// TIA Portal V20 export
DATA_BLOCK "InstCallEquipment"   // DB137
{ DB_Accessible_From_OPC_UA := 'FALSE' }
AUTHOR : ERsystem_FA2_DH. Kim
// stored: AssignedProDiagFB Unit1.Em7.ProDiag, DBAccessibleFromOPCUA false, DBAccessibleFromWebserver false, InstanceOfName Unit1.Em7.CallEquipment, InstanceOfType FB, Namespace Unit1.Em7
"Unit1.Em7.CallEquipment"
   // VAR_INPUT
   //    ZoneOperationEnable { ExternalWritable := 'False'} : "LWONIK_typeSafetyZoneManualOperation";
   // END_VAR
   // VAR_IN_OUT
   //    unitStatus : "LAF_typeUnitStatus";
   //    emFeedback : "LUC_typeEmFeedback";
   //    unitAlarmDB : "LAF_typeAlarms";
   // END_VAR
   // VAR
   //    instSequenceSepaClamp { ExternalAccessible := 'False'; ExternalVisible := 'False'; ExternalWritable := 'False'} : "Unit1.Em7.Sequence_1_SepaClamp";
   //    instSequenceSepaGripper { ExternalAccessible := 'False'; ExternalVisible := 'False'; ExternalWritable := 'False'} : "Unit1.Em7.Sequence_2_SepaGripper";
   //    instSequenceJellyRollWinder { ExternalAccessible := 'False'; ExternalVisible := 'False'; ExternalWritable := 'False'} : "Unit1.Em7.Sequence_3_JellyRollWinder";
   //    instSepaClampHomeJob1 { S7_SetPoint := 'True'} : "LAF_SelectJob";
   //    instSepaClampLoadJob2 { S7_SetPoint := 'True'} : "LAF_SelectJob";
   //    instSepaClampUnloadJob3 { S7_SetPoint := 'True'} : "LAF_SelectJob";
   //    instSepaClampUnloadCamJob10 { S7_SetPoint := 'True'} : "LAF_SelectJob";
   //    instSepaClampUnloadStopSyncJob11 { S7_SetPoint := 'True'} : "LAF_SelectJob";
   //    instSepaClampUnloadReturnJob12 { S7_SetPoint := 'True'} : "LAF_SelectJob";
   //    instSepaGripperHomeJob1 { S7_SetPoint := 'True'} : "LAF_SelectJob";
   //    instSepaGripperGripReadyJob2 { S7_SetPoint := 'True'} : "LAF_SelectJob";
   //    instSepaGripperGripSepaTailJob3 { S7_SetPoint := 'True'} : "LAF_SelectJob";
   //    instSepaGripperWinderMoveJob4 { S7_SetPoint := 'True'} : "LAF_SelectJob";
   //    instSepaGripperJellyRollUnGripJob5 { S7_SetPoint := 'True'} : "LAF_SelectJob";
   //    instSepaGripperJellyRollGripJob6 { S7_SetPoint := 'True'} : "LAF_SelectJob";
   //    instSepaGripperUnloadReadyJob7 { S7_SetPoint := 'True'} : "LAF_SelectJob";
   //    instSepaGripperUnloadJob8 { S7_SetPoint := 'True'} : "LAF_SelectJob";
   //    instSepaGripperReturnJob9 { S7_SetPoint := 'True'} : "LAF_SelectJob";
   //    instSepaGripperGripReadyJob11 { S7_SetPoint := 'True'} : "LAF_SelectJob";
   //    instSepaGripperLoadToStackTableJob12 { S7_SetPoint := 'True'} : "LAF_SelectJob";
   //    instSepaGripperUnLoadToJellyRollWinderJob14 { S7_SetPoint := 'True'} : "LAF_SelectJob";
   //    instSepaGripperLoadToJellyRollWinderJob15 { S7_SetPoint := 'True'} : "LAF_SelectJob";
   //    instSepaGripperUnloadToInspectionJob17 { S7_SetPoint := 'True'} : "LAF_SelectJob";
   //    instSepaGripperReturnJob18 { S7_SetPoint := 'True'} : "LAF_SelectJob";
   //    instJellyRollWinderHomeJob1 { S7_SetPoint := 'True'} : "LAF_SelectJob";
   //    instJellyRollWinderLoadJob2 { S7_SetPoint := 'True'} : "LAF_SelectJob";
   //    instJellyRollWinderWinding1Job3 { S7_SetPoint := 'True'} : "LAF_SelectJob";
   //    instJellyRollWinderPusherReadyJob4 { S7_SetPoint := 'True'} : "LAF_SelectJob";
   //    instJellyRollWinderWinding2Job5 { S7_SetPoint := 'True'} : "LAF_SelectJob";
   //    instJellyRollWinderUnloadJob6 { S7_SetPoint := 'True'} : "LAF_SelectJob";
   //    instJellyRollWinderCamWinding1stJob10 { S7_SetPoint := 'True'} : "LAF_SelectJob";
   //    instJellyRollWinderCamPusherReadyJob11 { S7_SetPoint := 'True'} : "LAF_SelectJob";
   //    instJellyRollWinderCamStartSyncJob12 { S7_SetPoint := 'True'} : "LAF_SelectJob";
   //    instJellyRollWinderCamWinding2ndJob13 { S7_SetPoint := 'True'} : "LAF_SelectJob";
   //    instJellyRollWinderCamStopSyncJob14 { S7_SetPoint := 'True'} : "LAF_SelectJob";
   //    instCmSepaClampDetectSensor { ExternalAccessible := 'False'; ExternalVisible := 'False'; ExternalWritable := 'False'} : "LBC_DigitalSignalCn";
   //    instCmSepaGripperDetectSensor { ExternalAccessible := 'False'; ExternalVisible := 'False'; ExternalWritable := 'False'} : "LBC_DigitalSignalCn";
   //    instCmJrWinderDetectSensor { ExternalAccessible := 'False'; ExternalVisible := 'False'; ExternalWritable := 'False'} : "LBC_DigitalSignalCn";
   //    instCmSepaElectrodeDetectSensor { ExternalAccessible := 'False'; ExternalVisible := 'False'; ExternalWritable := 'False'} : "LBC_DigitalSignalCn";
   //    instCmSepaClampSafetyPinDetectSensor { ExternalAccessible := 'False'; ExternalVisible := 'False'; ExternalWritable := 'False'} : "LBC_DigitalSignalCn";
   //    instCmSepaGripperSafetyPinDetectSensor { ExternalAccessible := 'False'; ExternalVisible := 'False'; ExternalWritable := 'False'} : "LBC_DigitalSignalCn";
   //    instCmSepaClampnCutterAxisX { ExternalAccessible := 'False'; ExternalVisible := 'False'; ExternalWritable := 'False'} : "LBC_Axis64Pos_TecPlcCn";
   //    instCmSepaClampnCutterAxisZ { ExternalAccessible := 'False'; ExternalVisible := 'False'; ExternalWritable := 'False'} : "LBC_Axis64Pos_TecPlcCn";
   //    instCmSepaGripperAxisX { ExternalAccessible := 'False'; ExternalVisible := 'False'; ExternalWritable := 'False'} : "LBC_Axis64Pos_TecPlcCn";
   //    instCmSepaGripperAxisZ { ExternalAccessible := 'False'; ExternalVisible := 'False'; ExternalWritable := 'False'} : "LBC_Axis64Pos_TecPlcCn";
   //    instCmSepaGripperAxisC { ExternalAccessible := 'False'; ExternalVisible := 'False'; ExternalWritable := 'False'} : "LBC_Axis64Pos_TecPlcCn";
   //    instCmJRWinderRearAxisY { ExternalAccessible := 'False'; ExternalVisible := 'False'; ExternalWritable := 'False'} : "LBC_Axis64Pos_TecPlcCn";
   //    instCmJRWinderFrontAxisY { ExternalAccessible := 'False'; ExternalVisible := 'False'; ExternalWritable := 'False'} : "LBC_Axis64Pos_TecPlcCn";
   //    instCmJRWinderAxisB { ExternalAccessible := 'False'; ExternalVisible := 'False'; ExternalWritable := 'False'} : "LBC_Axis64Pos_TecPlcCn";
   //    instCmJRPusherAxisZ { ExternalAccessible := 'False'; ExternalVisible := 'False'; ExternalWritable := 'False'} : "LBC_Axis64Pos_TecPlcCn";
   //    instInterlockSepaClampnCutterAxisX { S7_SetPoint := 'True'} : "LER_Axis64Pos_InterlockSummary";
   //    instInterlockSepaClampnCutterAxisZ { S7_SetPoint := 'True'} : "LER_Axis64Pos_InterlockSummary";
   //    instInterlockSepaGripperAxisX { S7_SetPoint := 'True'} : "LER_Axis64Pos_InterlockSummary";
   //    instInterlockSepaGripperAxisZ { S7_SetPoint := 'True'} : "LER_Axis64Pos_InterlockSummary";
   //    instInterlockSepaGripperAxisC { S7_SetPoint := 'True'} : "LER_Axis64Pos_InterlockSummary";
   //    instInterlockJRWinderRearAxisY { S7_SetPoint := 'True'} : "LER_Axis64Pos_InterlockSummary";
   //    instInterlockJRWinderFrontAxisY { S7_SetPoint := 'True'} : "LER_Axis64Pos_InterlockSummary";
   //    instInterlockJRWinderAxisB { S7_SetPoint := 'True'} : "LER_Axis64Pos_InterlockSummary";
   //    instInterlockJRPusherAxisZ { S7_SetPoint := 'True'} : "LER_Axis64Pos_InterlockSummary";
   //    instSepaClampAxisXCalculateCam { S7_SetPoint := 'True'} : "Unit1.Em7.SepaClampXCalculateCam";
   //    instSepaClampAxisZCalculateCam { S7_SetPoint := 'True'} : "Unit1.Em7.SepaClampZCalculateCam";
   //    instJRPusherAxisZCalculateCam { S7_SetPoint := 'True'} : "Unit1.Em7.PusherRollerZCalculateCam";
   //    instSepaClampAxisXMCCamIn { S7_SetPoint := 'True'} : MC_CAMIN;
   //    instSepaClampAxisZMCCamIn { S7_SetPoint := 'True'} : MC_CAMIN;
   //    instJRPusherAxisZMCCamIn { S7_SetPoint := 'True'} : MC_CAMIN;
   //    instCmSepaCutterUpDown { ExternalAccessible := 'False'; ExternalVisible := 'False'; ExternalWritable := 'False'} : "LBC_TwoWayActuatorCn";
   //    instCmSepaClampTopUpDown { ExternalAccessible := 'False'; ExternalVisible := 'False'; ExternalWritable := 'False'} : "LBC_TwoWayActuatorCn";
   //    instCmSepaClampBottomUpDown { ExternalAccessible := 'False'; ExternalVisible := 'False'; ExternalWritable := 'False'} : "LBC_TwoWayActuatorCn";
   //    instCmStackGripperOpenClose { ExternalAccessible := 'False'; ExternalVisible := 'False'; ExternalWritable := 'False'} : "LBC_TwoWayActuatorCn";
   //    instCmStackGripperFwdBwd { ExternalAccessible := 'False'; ExternalVisible := 'False'; ExternalWritable := 'False'} : "LBC_TwoWayActuatorCn";
   //    instCmJRWinderClampTopRearUpDown { ExternalAccessible := 'False'; ExternalVisible := 'False'; ExternalWritable := 'False'} : "LBC_TwoWayActuatorCn";
   //    instCmJRWinderClampBtmRearUpDown { ExternalAccessible := 'False'; ExternalVisible := 'False'; ExternalWritable := 'False'} : "LBC_TwoWayActuatorCn";
   //    instCmJRWinderClampTopFrontUpDown { ExternalAccessible := 'False'; ExternalVisible := 'False'; ExternalWritable := 'False'} : "LBC_TwoWayActuatorCn";
   //    instCmJRWinderClampBtmFrontUpDown { ExternalAccessible := 'False'; ExternalVisible := 'False'; ExternalWritable := 'False'} : "LBC_TwoWayActuatorCn";
   //    instCmPusherRollerFwdBwd { ExternalAccessible := 'False'; ExternalVisible := 'False'; ExternalWritable := 'False'} : "LBC_TwoWayActuatorCn";
   //    instManageAlarms { ExternalAccessible := 'False'; ExternalVisible := 'False'; ExternalWritable := 'False'} : "LAF_ManageAlarms";
   //    instEventsPFE { ExternalAccessible := 'False'; ExternalVisible := 'False'; ExternalWritable := 'False'} : "Unit1.Em7.EventsPFE";
   //    instLER_BrakeTestSepaClampNCutterAxisZ : "LER_BrakeTest";
   //    instLER_BrakeTestSepaGripperAxisZ { S7_SetPoint := 'True'} : "LER_BrakeTest";
   //    instLER_BrakeTestJRPusherAxisZ { S7_SetPoint := 'True'} : "LER_BrakeTest";
   //    statUnitStatus { ExternalAccessible := 'False'; ExternalVisible := 'False'; ExternalWritable := 'False'} : "LAF_typeUnitStatus";
   //    statSlmStatus : Struct
   //       running { ExternalWritable := 'False'} : Bool;
   //       powerOff { ExternalWritable := 'False'} : Bool;
   //    END_STRUCT;
   //    statAllBrakeTest { ExternalWritable := 'False'} : "LER_typeBrakeTestUnitCommands";
   //    statTonTime { ExternalAccessible := 'False'; ExternalVisible := 'False'; ExternalWritable := 'False'} : Array[0..1999] of TON_TIME;
   //    statTofTime { ExternalAccessible := 'False'; ExternalVisible := 'False'; ExternalWritable := 'False'} : Array[0..99] of TOF_TIME;
   //    statPulse { ExternalAccessible := 'False'; ExternalVisible := 'False'; ExternalWritable := 'False'} : Struct
   //       miscellaneous : Array[0..99] of Bool;
   //       workingDone : Struct
   //          sepaClamp : Array[0..99] of Bool;
   //          sepaGripper : Array[0..99] of Bool;
   //          winder : Array[0..99] of Bool;
   //       END_STRUCT;
   //       axisEnable : Array[0..99] of Bool;
   //       brakeTest : Array[0..99] of Bool;
   //    END_STRUCT;
   //    statEnableManualCmds { ExternalAccessible := 'False'; ExternalVisible := 'False'; ExternalWritable := 'False'} : Bool;
   //    scan_on : Bool;
   //    "*** Interlock Axis ***" { ExternalAccessible := 'False'; ExternalVisible := 'False'; ExternalWritable := 'False'} : Bool;
   //    instSepaClampnCutterAxisX_CW { S7_SetPoint := 'True'} : "Jog.LER_Axis";
   //    instSepaClampnCutterAxisX_CCW { S7_SetPoint := 'True'} : "Jog.LER_Axis";
   //    instSepaClampnCutterAxisX_Home { S7_SetPoint := 'True'} : "Homing.LER_Axis";
   //    instSepaClampnCutterAxisX_Position { S7_SetPoint := 'True'} : Array[0..6] of "Position.LER_Axis";
   //    instSepaClampnCutterAxisZ_CW { S7_SetPoint := 'True'} : "Jog.LER_Axis";
   //    instSepaClampnCutterAxisZ_CCW { S7_SetPoint := 'True'} : "Jog.LER_Axis";
   //    instSepaClampnCutterAxisZ_Home { S7_SetPoint := 'True'} : "Homing.LER_Axis";
   //    instSepaClampnCutterAxisZ_Position { S7_SetPoint := 'True'} : Array[0..6] of "Position.LER_Axis";
   //    instSepaGripperAxisX_CW { S7_SetPoint := 'True'} : "Jog.LER_Axis";
   //    instSepaGripperAxisX_CCW { S7_SetPoint := 'True'} : "Jog.LER_Axis";
   //    instSepaGripperAxisX_Home { S7_SetPoint := 'True'} : "Homing.LER_Axis";
   //    instSepaGripperAxisX_Position { S7_SetPoint := 'True'} : Array[0..15] of "Position.LER_Axis";
   //    instSepaGripperAxisZ_CW { S7_SetPoint := 'True'} : "Jog.LER_Axis";
   //    instSepaGripperAxisZ_CCW { S7_SetPoint := 'True'} : "Jog.LER_Axis";
   //    instSepaGripperAxisZ_Home { S7_SetPoint := 'True'} : "Homing.LER_Axis";
   //    instSepaGripperAxisZ_Position { S7_SetPoint := 'True'} : Array[0..6] of "Position.LER_Axis";
   //    instSepaGripperAxisC_CW { S7_SetPoint := 'True'} : "Jog.LER_Axis";
   //    instSepaGripperAxisC_CCW { S7_SetPoint := 'True'} : "Jog.LER_Axis";
   //    instSepaGripperAxisC_Home { S7_SetPoint := 'True'} : "Homing.LER_Axis";
   //    instSepaGripperAxisC_Position { S7_SetPoint := 'True'} : Array[0..6] of "Position.LER_Axis";
   //    instJRWinderRearAxisY_CW { S7_SetPoint := 'True'} : "Jog.LER_Axis";
   //    instJRWinderRearAxisY_CCW { S7_SetPoint := 'True'} : "Jog.LER_Axis";
   //    instJRWinderRearAxisY_Home { S7_SetPoint := 'True'} : "Homing.LER_Axis";
   //    instJRWinderRearAxisY_Position { S7_SetPoint := 'True'} : Array[0..6] of "Position.LER_Axis";
   //    instJRWinderFrontAxisY_CW { S7_SetPoint := 'True'} : "Jog.LER_Axis";
   //    instJRWinderFrontAxisY_CCW { S7_SetPoint := 'True'} : "Jog.LER_Axis";
   //    instJRWinderFrontAxisY_Home { S7_SetPoint := 'True'} : "Homing.LER_Axis";
   //    instJRWinderFrontAxisY_Position { S7_SetPoint := 'True'} : Array[0..6] of "Position.LER_Axis";
   //    instJRWinderAxisB_CW { S7_SetPoint := 'True'} : "Jog.LER_Axis";
   //    instJRWinderAxisB_CCW { S7_SetPoint := 'True'} : "Jog.LER_Axis";
   //    instJRWinderAxisB_Home { S7_SetPoint := 'True'} : "Homing.LER_Axis";
   //    instJRWinderAxisB_Position { S7_SetPoint := 'True'} : Array[0..8] of "Position.LER_Axis";
   //    instJRPusherAxisZ_CW { S7_SetPoint := 'True'} : "Jog.LER_Axis";
   //    instJRPusherAxisZ_CCW { S7_SetPoint := 'True'} : "Jog.LER_Axis";
   //    instJRPusherAxisZ_Home { S7_SetPoint := 'True'} : "Homing.LER_Axis";
   //    instJRPusherAxisZ_Position { S7_SetPoint := 'True'} : Array[0..6] of "Position.LER_Axis";
   //    "*** Interlock Actuator ******" { ExternalAccessible := 'False'; ExternalVisible := 'False'; ExternalWritable := 'False'} : Bool;
   //    instCmSepaCutterUpDownInterlock : Array[0..1] of "Cylinder.LER_Actuator";
   //    instCmSepaClampTopUpDownInterlock { S7_SetPoint := 'True'} : Array[0..1] of "Cylinder.LER_Actuator";
   //    instCmSepaClampBottomUpDownInterlock { S7_SetPoint := 'True'} : Array[0..1] of "Cylinder.LER_Actuator";
   //    instCmStackGripperOpenCloseInterlock { S7_SetPoint := 'True'} : Array[0..1] of "Cylinder.LER_Actuator";
   //    instCmStackGripperFwdBwdInterlock { S7_SetPoint := 'True'} : Array[0..1] of "Cylinder.LER_Actuator";
   //    instCmJRWinderClampTopRearUpDownInterlock { S7_SetPoint := 'True'} : Array[0..1] of "Cylinder.LER_Actuator";
   //    instCmJRWinderClampBtmRearUpDownInterlock { S7_SetPoint := 'True'} : Array[0..1] of "Cylinder.LER_Actuator";
   //    instCmJRWinderClampTopFrontUpDownInterlock { S7_SetPoint := 'True'} : Array[0..1] of "Cylinder.LER_Actuator";
   //    instCmJRWinderClampBtmFrontUpDownInterlock { S7_SetPoint := 'True'} : Array[0..1] of "Cylinder.LER_Actuator";
   //    instCmPusherRollerFwdBwdInterlock { S7_SetPoint := 'True'} : Array[0..1] of "Cylinder.LER_Actuator";
   //    Tracking_07 { S7_SetPoint := 'True'} : "Unit1.Em7.PartData";
   //    AXIS34 : "LER_CM_Name";
   //    AXIS39 : "LER_CM_Name";
   //    Cylinder38 : "LER_CM_Name";
   //    Cylinder43 : "LER_CM_Name";
   //    citi_Ptrig : Array[0..20] of Bool;
   //    citiTon : Array[0..20] of TON_TIME;
   //    citi : Time;
   //    citiTest : Array[0..20] of Bool;
   // END_VAR
BEGIN
   ZoneOperationEnable.autoStartEnable := FALSE;
   ZoneOperationEnable.doorLockEnable := TRUE;
   ZoneOperationEnable.doorUnlockEnable := TRUE;
   ZoneOperationEnable.rc_AutoEnable := FALSE;
   ZoneOperationEnable.rc_RollChangeEnable := FALSE;
   ZoneOperationEnable.rc_DoorLockEnable := TRUE;
   ZoneOperationEnable.rc_DoorUnlockEnable := TRUE;
   ZoneOperationEnable.hmiOperationEnable := TRUE;
   ZoneOperationEnable.phmiOperationEnable := FALSE;
   instSequenceSepaClamp.statSelectedJobNumber := 0;
   instSequenceSepaClamp.instSequenceLADStatus.parentReferenceDesignator := WSTRING#'';
   instSequenceSepaClamp.instSequenceLADStatus.idleStep := 1;
   instSequenceSepaClamp.instSequenceLADStatus.stoppedStep := 9001;
   instSequenceSepaClamp.instSequenceLADStatus.setJobNumber := 0;
   instSequenceSepaClamp.instSequenceLADStatus.activeJobNumber := 0;
   instSequenceSepaClamp.instSequenceLADStatus.previousCycleJobNumber := 0;
   instSequenceSepaClamp.instSequenceLADStatus.statCurrentJob := 0;
   instSequenceSepaClamp.instSequenceLADStatus.statStepComplete := FALSE;
   instSequenceSepaClamp.instSequenceLADControl.idleStep := 1;
   instSequenceSepaClamp.instSequenceLADControl.stoppedStep := 9001;
   instSequenceSepaClamp.instSequenceLADControl.resetJobs := FALSE;
   instSequenceSepaClamp.instSequenceLADControl.statMemInit := FALSE;
   instSequenceSepaClamp.instSequenceLADControl.statMemImmediateStop := FALSE;
   instSequenceSepaClamp.instSequenceLADControl.statMemNextStep1 := FALSE;
   instSequenceSepaClamp.instSequenceLADControl.statMemNextStep2 := FALSE;
   instSequenceSepaClamp.instSequenceLADControl.statMemNextStep3 := FALSE;
   instSequenceSepaClamp.instSequenceLADControl.statFirstCycleInit := FALSE;
   instCmSepaClampDetectSensor.enable := TRUE;
   instCmSepaClampDetectSensor.parentReferenceDesignator := WSTRING#'';
   instCmSepaClampDetectSensor.digitalValue := FALSE;
   instCmSepaClampDetectSensor.simulatedDigitalValue := FALSE;
   instCmSepaClampDetectSensor.statProcessValues.enable := TRUE;
   instCmSepaClampDetectSensor.statProcessValues.referenceDesignator := WSTRING#'DigitalSignal';
   instCmSepaClampDetectSensor.statProcessValues.simulation := FALSE;
   instCmSepaClampDetectSensor.statProcessValues.processValue := FALSE;
   instCmSepaClampDetectSensor.statProcessValues.error := FALSE;
   instCmSepaClampDetectSensor.statProcessValues.status := 16#0000;
   instCmSepaClampDetectSensor.statDiagnostics.status := 16#0000;
   instCmSepaClampDetectSensor.statDiagnostics.subfunctionStatus := 16#0000;
   instCmSepaClampDetectSensor.statDiagnostics.stateNumber := 0;
   instCmSepaClampDetectSensor.statEmptyDiagnostics.status := 16#0000;
   instCmSepaClampDetectSensor.statEmptyDiagnostics.subfunctionStatus := 16#0000;
   instCmSepaClampDetectSensor.statEmptyDiagnostics.stateNumber := 0;
   instCmSepaClampDetectSensor.instOnDelay.PT := T#0MS;
   instCmSepaClampDetectSensor.instOnDelay.IN := FALSE;
   instCmSepaClampDetectSensor.instOffDelay.PT := T#0MS;
   instCmSepaClampDetectSensor.instOffDelay.IN := FALSE;
   instCmSepaClampDetectSensor.statDisableAlarms := FALSE;
   instCmSepaClampDetectSensor.statErrorState := 16#0000;
   instCmSepaClampDetectSensor.statFirstCall := FALSE;
   instCmSepaClampDetectSensor.statResetPrevious := FALSE;
   instCmSepaClampDetectSensor.statEnablePrevious := TRUE;
   instCmSepaClampDetectSensor.statProcessValuePrevious := FALSE;
   instCmSepaGripperDetectSensor.enable := TRUE;
   instCmSepaGripperDetectSensor.parentReferenceDesignator := WSTRING#'';
   instCmSepaGripperDetectSensor.digitalValue := TRUE;
   instCmSepaGripperDetectSensor.simulatedDigitalValue := FALSE;
   instCmSepaGripperDetectSensor.statProcessValues.enable := TRUE;
   instCmSepaGripperDetectSensor.statProcessValues.referenceDesignator := WSTRING#'DigitalSignal';
   instCmSepaGripperDetectSensor.statProcessValues.simulation := FALSE;
   instCmSepaGripperDetectSensor.statProcessValues.processValue := TRUE;
   instCmSepaGripperDetectSensor.statProcessValues.error := FALSE;
   instCmSepaGripperDetectSensor.statProcessValues.status := 16#0000;
   instCmSepaGripperDetectSensor.statDiagnostics.status := 16#0000;
   instCmSepaGripperDetectSensor.statDiagnostics.subfunctionStatus := 16#0000;
   instCmSepaGripperDetectSensor.statDiagnostics.stateNumber := 0;
   instCmSepaGripperDetectSensor.statEmptyDiagnostics.status := 16#0000;
   instCmSepaGripperDetectSensor.statEmptyDiagnostics.subfunctionStatus := 16#0000;
   instCmSepaGripperDetectSensor.statEmptyDiagnostics.stateNumber := 0;
   instCmSepaGripperDetectSensor.instOnDelay.PT := T#0MS;
   instCmSepaGripperDetectSensor.instOnDelay.IN := FALSE;
   instCmSepaGripperDetectSensor.instOffDelay.PT := T#0MS;
   instCmSepaGripperDetectSensor.instOffDelay.IN := FALSE;
   instCmSepaGripperDetectSensor.statDisableAlarms := FALSE;
   instCmSepaGripperDetectSensor.statErrorState := 16#0000;
   instCmSepaGripperDetectSensor.statFirstCall := FALSE;
   instCmSepaGripperDetectSensor.statResetPrevious := FALSE;
   instCmSepaGripperDetectSensor.statEnablePrevious := TRUE;
   instCmSepaGripperDetectSensor.statProcessValuePrevious := TRUE;
   instCmJrWinderDetectSensor.enable := TRUE;
   instCmJrWinderDetectSensor.parentReferenceDesignator := WSTRING#'';
   instCmJrWinderDetectSensor.digitalValue := FALSE;
   instCmJrWinderDetectSensor.simulatedDigitalValue := FALSE;
   instCmJrWinderDetectSensor.statProcessValues.enable := TRUE;
   instCmJrWinderDetectSensor.statProcessValues.referenceDesignator := WSTRING#'DigitalSignal';
   instCmJrWinderDetectSensor.statProcessValues.simulation := FALSE;
   instCmJrWinderDetectSensor.statProcessValues.processValue := FALSE;
   instCmJrWinderDetectSensor.statProcessValues.error := FALSE;
   instCmJrWinderDetectSensor.statProcessValues.status := 16#0000;
   instCmJrWinderDetectSensor.statDiagnostics.status := 16#0000;
   instCmJrWinderDetectSensor.statDiagnostics.subfunctionStatus := 16#0000;
   instCmJrWinderDetectSensor.statDiagnostics.stateNumber := 0;
   instCmJrWinderDetectSensor.statEmptyDiagnostics.status := 16#0000;
   instCmJrWinderDetectSensor.statEmptyDiagnostics.subfunctionStatus := 16#0000;
   instCmJrWinderDetectSensor.statEmptyDiagnostics.stateNumber := 0;
   instCmJrWinderDetectSensor.instOnDelay.PT := T#0MS;
   instCmJrWinderDetectSensor.instOnDelay.IN := FALSE;
   instCmJrWinderDetectSensor.instOffDelay.PT := T#0MS;
   instCmJrWinderDetectSensor.instOffDelay.IN := FALSE;
   instCmJrWinderDetectSensor.statDisableAlarms := FALSE;
   instCmJrWinderDetectSensor.statErrorState := 16#0000;
   instCmJrWinderDetectSensor.statFirstCall := FALSE;
   instCmJrWinderDetectSensor.statResetPrevious := FALSE;
   instCmJrWinderDetectSensor.statEnablePrevious := TRUE;
   instCmJrWinderDetectSensor.statProcessValuePrevious := FALSE;
   instCmSepaElectrodeDetectSensor.enable := TRUE;
   instCmSepaElectrodeDetectSensor.parentReferenceDesignator := WSTRING#'';
   instCmSepaElectrodeDetectSensor.digitalValue := FALSE;
   instCmSepaElectrodeDetectSensor.simulatedDigitalValue := FALSE;
   instCmSepaElectrodeDetectSensor.statProcessValues.enable := TRUE;
   instCmSepaElectrodeDetectSensor.statProcessValues.referenceDesignator := WSTRING#'DigitalSignal';
   instCmSepaElectrodeDetectSensor.statProcessValues.simulation := FALSE;
   instCmSepaElectrodeDetectSensor.statProcessValues.processValue := FALSE;
   instCmSepaElectrodeDetectSensor.statProcessValues.error := FALSE;
   instCmSepaElectrodeDetectSensor.statProcessValues.status := 16#0000;
   instCmSepaElectrodeDetectSensor.statDiagnostics.status := 16#0000;
   instCmSepaElectrodeDetectSensor.statDiagnostics.subfunctionStatus := 16#0000;
   instCmSepaElectrodeDetectSensor.statDiagnostics.stateNumber := 0;
   instCmSepaElectrodeDetectSensor.statEmptyDiagnostics.status := 16#0000;
   instCmSepaElectrodeDetectSensor.statEmptyDiagnostics.subfunctionStatus := 16#0000;
   instCmSepaElectrodeDetectSensor.statEmptyDiagnostics.stateNumber := 0;
   instCmSepaElectrodeDetectSensor.instOnDelay.PT := T#0MS;
   instCmSepaElectrodeDetectSensor.instOnDelay.IN := FALSE;
   instCmSepaElectrodeDetectSensor.instOffDelay.PT := T#0MS;
   instCmSepaElectrodeDetectSensor.instOffDelay.IN := FALSE;
   instCmSepaElectrodeDetectSensor.statDisableAlarms := FALSE;
   instCmSepaElectrodeDetectSensor.statErrorState := 16#0000;
   instCmSepaElectrodeDetectSensor.statFirstCall := FALSE;
   instCmSepaElectrodeDetectSensor.statResetPrevious := FALSE;
   instCmSepaElectrodeDetectSensor.statEnablePrevious := TRUE;
   instCmSepaElectrodeDetectSensor.statProcessValuePrevious := FALSE;
   instCmSepaClampSafetyPinDetectSensor.enable := TRUE;
   instCmSepaClampSafetyPinDetectSensor.parentReferenceDesignator := WSTRING#'';
   instCmSepaClampSafetyPinDetectSensor.digitalValue := TRUE;
   instCmSepaClampSafetyPinDetectSensor.simulatedDigitalValue := FALSE;
   instCmSepaClampSafetyPinDetectSensor.statProcessValues.enable := TRUE;
   instCmSepaClampSafetyPinDetectSensor.statProcessValues.referenceDesignator := WSTRING#'DigitalSignal';
   instCmSepaClampSafetyPinDetectSensor.statProcessValues.simulation := FALSE;
   instCmSepaClampSafetyPinDetectSensor.statProcessValues.processValue := TRUE;
   instCmSepaClampSafetyPinDetectSensor.statProcessValues.error := FALSE;
   instCmSepaClampSafetyPinDetectSensor.statProcessValues.status := 16#0000;
   instCmSepaClampSafetyPinDetectSensor.statDiagnostics.status := 16#0000;
   instCmSepaClampSafetyPinDetectSensor.statDiagnostics.subfunctionStatus := 16#0000;
   instCmSepaClampSafetyPinDetectSensor.statDiagnostics.stateNumber := 0;
   instCmSepaClampSafetyPinDetectSensor.statEmptyDiagnostics.status := 16#0000;
   instCmSepaClampSafetyPinDetectSensor.statEmptyDiagnostics.subfunctionStatus := 16#0000;
   instCmSepaClampSafetyPinDetectSensor.statEmptyDiagnostics.stateNumber := 0;
   instCmSepaClampSafetyPinDetectSensor.instOnDelay.PT := T#0MS;
   instCmSepaClampSafetyPinDetectSensor.instOnDelay.IN := FALSE;
   instCmSepaClampSafetyPinDetectSensor.instOffDelay.PT := T#0MS;
   instCmSepaClampSafetyPinDetectSensor.instOffDelay.IN := FALSE;
   instCmSepaClampSafetyPinDetectSensor.statDisableAlarms := FALSE;
   instCmSepaClampSafetyPinDetectSensor.statErrorState := 16#0000;
   instCmSepaClampSafetyPinDetectSensor.statFirstCall := FALSE;
   instCmSepaClampSafetyPinDetectSensor.statResetPrevious := FALSE;
   instCmSepaClampSafetyPinDetectSensor.statEnablePrevious := TRUE;
   instCmSepaClampSafetyPinDetectSensor.statProcessValuePrevious := TRUE;
   instCmSepaGripperSafetyPinDetectSensor.enable := FALSE;
   instCmSepaGripperSafetyPinDetectSensor.parentReferenceDesignator := WSTRING#'';
   instCmSepaGripperSafetyPinDetectSensor.digitalValue := FALSE;
   instCmSepaGripperSafetyPinDetectSensor.simulatedDigitalValue := FALSE;
   instCmSepaGripperSafetyPinDetectSensor.statProcessValues.enable := FALSE;
   instCmSepaGripperSafetyPinDetectSensor.statProcessValues.referenceDesignator := WSTRING#'';
   instCmSepaGripperSafetyPinDetectSensor.statProcessValues.simulation := FALSE;
   instCmSepaGripperSafetyPinDetectSensor.statProcessValues.processValue := FALSE;
   instCmSepaGripperSafetyPinDetectSensor.statProcessValues.error := FALSE;
   instCmSepaGripperSafetyPinDetectSensor.statProcessValues.status := 16#0000;
   instCmSepaGripperSafetyPinDetectSensor.statDiagnostics.status := 16#7000;
   instCmSepaGripperSafetyPinDetectSensor.statDiagnostics.subfunctionStatus := 16#0000;
   instCmSepaGripperSafetyPinDetectSensor.statDiagnostics.stateNumber := 0;
   instCmSepaGripperSafetyPinDetectSensor.statEmptyDiagnostics.status := 16#0000;
   instCmSepaGripperSafetyPinDetectSensor.statEmptyDiagnostics.subfunctionStatus := 16#0000;
   instCmSepaGripperSafetyPinDetectSensor.statEmptyDiagnostics.stateNumber := 0;
   instCmSepaGripperSafetyPinDetectSensor.instOnDelay.PT := T#0MS;
   instCmSepaGripperSafetyPinDetectSensor.instOnDelay.IN := FALSE;
   instCmSepaGripperSafetyPinDetectSensor.instOffDelay.PT := T#0MS;
   instCmSepaGripperSafetyPinDetectSensor.instOffDelay.IN := FALSE;
   instCmSepaGripperSafetyPinDetectSensor.statDisableAlarms := FALSE;
   instCmSepaGripperSafetyPinDetectSensor.statErrorState := 16#7000;
   instCmSepaGripperSafetyPinDetectSensor.statFirstCall := TRUE;
   instCmSepaGripperSafetyPinDetectSensor.statResetPrevious := FALSE;
   instCmSepaGripperSafetyPinDetectSensor.statEnablePrevious := FALSE;
   instCmSepaGripperSafetyPinDetectSensor.statProcessValuePrevious := FALSE;
   instCmSepaCutterUpDown.enable := TRUE;
   instCmSepaCutterUpDown.parentReferenceDesignator := WSTRING#'';
   instCmSepaCutterUpDown.feedbackHomePos := FALSE;
   instCmSepaCutterUpDown.feedbackWorkPos := TRUE;
   instCmSepaCutterUpDown.enableManualCmds := TRUE;
   instCmSepaCutterUpDown.interlockWorkPos := TRUE;
   instCmSepaCutterUpDown.interlockHomePos := TRUE;
   instCmSepaCutterUpDown.goToHomePos := FALSE;
   instCmSepaCutterUpDown.goToWorkPos := FALSE;
   instCmSepaCutterUpDown.statProcessValues.enable := TRUE;
   instCmSepaCutterUpDown.statProcessValues.referenceDesignator := WSTRING#'SepaCutterUpDown';
   instCmSepaCutterUpDown.statProcessValues.commandHomePos := FALSE;
   instCmSepaCutterUpDown.statProcessValues.commandWorkPos := FALSE;
   instCmSepaCutterUpDown.statProcessValues.goToHomePos := FALSE;
   instCmSepaCutterUpDown.statProcessValues.goToWorkPos := FALSE;
   instCmSepaCutterUpDown.statProcessValues.inHomePos := FALSE;
   instCmSepaCutterUpDown.statProcessValues.inWorkPos := TRUE;
   instCmSepaCutterUpDown.statProcessValues.reset := FALSE;
   instCmSepaCutterUpDown.statProcessValues.enableManualCmds := TRUE;
   instCmSepaCutterUpDown.statProcessValues.error := FALSE;
   instCmSepaCutterUpDown.statProcessValues.interlockHomePos := TRUE;
   instCmSepaCutterUpDown.statProcessValues.interlockWorkPos := TRUE;
   instCmSepaCutterUpDown.statProcessValues.status := 16#7003;
   instCmSepaCutterUpDown.statProcessValues.interlockWarningWorkPos := FALSE;
   instCmSepaCutterUpDown.statProcessValues.interlockWarningHomePos := FALSE;
   instCmSepaCutterUpDown.statCurrentInputs.commandHomePos := FALSE;
   instCmSepaCutterUpDown.statCurrentInputs.commandWorkPos := FALSE;
   instCmSepaCutterUpDown.statCurrentInputs.reset := FALSE;
   instCmSepaCutterUpDown.statPreviousInputs.commandHomePos := FALSE;
   instCmSepaCutterUpDown.statPreviousInputs.commandWorkPos := FALSE;
   instCmSepaCutterUpDown.statPreviousInputs.reset := FALSE;
   instCmSepaCutterUpDown.statCurrentInterface.commandHomePos := FALSE;
   instCmSepaCutterUpDown.statCurrentInterface.commandWorkPos := FALSE;
   instCmSepaCutterUpDown.statCurrentInterface.reset := FALSE;
   instCmSepaCutterUpDown.statPreviousInterface.commandHomePos := FALSE;
   instCmSepaCutterUpDown.statPreviousInterface.commandWorkPos := FALSE;
   instCmSepaCutterUpDown.statPreviousInterface.reset := FALSE;
   instCmSepaCutterUpDown.statEmptyDiagnostics.status := 16#0000;
   instCmSepaCutterUpDown.statEmptyDiagnostics.subfunctionStatus := 16#0000;
   instCmSepaCutterUpDown.statEmptyDiagnostics.stateNumber := 0;
   instCmSepaCutterUpDown.instTimerReachPos.PT := T#0MS;
   instCmSepaCutterUpDown.instTimerReachPos.IN := FALSE;
   instCmSepaCutterUpDown.instTimerLeavePos.PT := T#0MS;
   instCmSepaCutterUpDown.instTimerLeavePos.IN := FALSE;
   instCmSepaCutterUpDown.instTimerDiscrepancyCheck.PT := T#0MS;
   instCmSepaCutterUpDown.instTimerDiscrepancyCheck.IN := FALSE;
   instCmSepaCutterUpDown.statDisableAlarms := FALSE;
   instCmSepaCutterUpDown.statDiagnostics.status := 16#7003;
   instCmSepaCutterUpDown.statDiagnostics.subfunctionStatus := 16#0000;
   instCmSepaCutterUpDown.statDiagnostics.stateNumber := 0;
   instCmSepaCutterUpDown.statEnablePrevious := TRUE;
   instCmSepaCutterUpDown.statFirstCall := FALSE;
   instCmSepaCutterUpDown.statResetPrevious := FALSE;
   instCmSepaCutterUpDown.statValid := TRUE;
   instCmSepaCutterUpDown.statBusy := TRUE;
   instCmSepaCutterUpDown.statError := FALSE;
   instCmSepaCutterUpDown.statInterlockWorkOff := FALSE;
   instCmSepaCutterUpDown.statInterlockHomeOff := FALSE;
   instCmSepaCutterUpDown.statFbState := 50;
   instCmSepaCutterUpDown.statFbStatePrevious := 50;
   instCmSepaCutterUpDown.statErrorUserCleared := FALSE;
   instCmSepaCutterUpDown.statErrorAutoCleared := FALSE;
   instCmSepaCutterUpDown.statErrorState := 16#0000;
   instCmSepaCutterUpDown.statDisablingCompleted := FALSE;
   instCmSepaCutterUpDown.statFeedbackHomePos := FALSE;
   instCmSepaCutterUpDown.statFeedbackWorkPos := TRUE;
   instCmSepaClampTopUpDown.enable := TRUE;
   instCmSepaClampTopUpDown.parentReferenceDesignator := WSTRING#'';
   instCmSepaClampTopUpDown.feedbackHomePos := FALSE;
   instCmSepaClampTopUpDown.feedbackWorkPos := TRUE;
   instCmSepaClampTopUpDown.enableManualCmds := TRUE;
   instCmSepaClampTopUpDown.interlockWorkPos := TRUE;
   instCmSepaClampTopUpDown.interlockHomePos := TRUE;
   instCmSepaClampTopUpDown.goToHomePos := FALSE;
   instCmSepaClampTopUpDown.goToWorkPos := FALSE;
   instCmSepaClampTopUpDown.statProcessValues.enable := TRUE;
   instCmSepaClampTopUpDown.statProcessValues.referenceDesignator := WSTRING#'SepaClampTopUpDown';
   instCmSepaClampTopUpDown.statProcessValues.commandHomePos := FALSE;
   instCmSepaClampTopUpDown.statProcessValues.commandWorkPos := FALSE;
   instCmSepaClampTopUpDown.statProcessValues.goToHomePos := FALSE;
   instCmSepaClampTopUpDown.statProcessValues.goToWorkPos := FALSE;
   instCmSepaClampTopUpDown.statProcessValues.inHomePos := FALSE;
   instCmSepaClampTopUpDown.statProcessValues.inWorkPos := TRUE;
   instCmSepaClampTopUpDown.statProcessValues.reset := FALSE;
   instCmSepaClampTopUpDown.statProcessValues.enableManualCmds := TRUE;
   instCmSepaClampTopUpDown.statProcessValues.error := FALSE;
   instCmSepaClampTopUpDown.statProcessValues.interlockHomePos := TRUE;
   instCmSepaClampTopUpDown.statProcessValues.interlockWorkPos := TRUE;
   instCmSepaClampTopUpDown.statProcessValues.status := 16#7003;
   instCmSepaClampTopUpDown.statProcessValues.interlockWarningWorkPos := FALSE;
   instCmSepaClampTopUpDown.statProcessValues.interlockWarningHomePos := FALSE;
   instCmSepaClampTopUpDown.statCurrentInputs.commandHomePos := FALSE;
   instCmSepaClampTopUpDown.statCurrentInputs.commandWorkPos := FALSE;
   instCmSepaClampTopUpDown.statCurrentInputs.reset := FALSE;
   instCmSepaClampTopUpDown.statPreviousInputs.commandHomePos := FALSE;
   instCmSepaClampTopUpDown.statPreviousInputs.commandWorkPos := FALSE;
   instCmSepaClampTopUpDown.statPreviousInputs.reset := FALSE;
   instCmSepaClampTopUpDown.statCurrentInterface.commandHomePos := FALSE;
   instCmSepaClampTopUpDown.statCurrentInterface.commandWorkPos := FALSE;
   instCmSepaClampTopUpDown.statCurrentInterface.reset := FALSE;
   instCmSepaClampTopUpDown.statPreviousInterface.commandHomePos := FALSE;
   instCmSepaClampTopUpDown.statPreviousInterface.commandWorkPos := FALSE;
   instCmSepaClampTopUpDown.statPreviousInterface.reset := FALSE;
   instCmSepaClampTopUpDown.statEmptyDiagnostics.status := 16#0000;
   instCmSepaClampTopUpDown.statEmptyDiagnostics.subfunctionStatus := 16#0000;
   instCmSepaClampTopUpDown.statEmptyDiagnostics.stateNumber := 0;
   instCmSepaClampTopUpDown.instTimerReachPos.PT := T#0MS;
   instCmSepaClampTopUpDown.instTimerReachPos.IN := FALSE;
   instCmSepaClampTopUpDown.instTimerLeavePos.PT := T#0MS;
   instCmSepaClampTopUpDown.instTimerLeavePos.IN := FALSE;
   instCmSepaClampTopUpDown.instTimerDiscrepancyCheck.PT := T#0MS;
   instCmSepaClampTopUpDown.instTimerDiscrepancyCheck.IN := FALSE;
   instCmSepaClampTopUpDown.statDisableAlarms := FALSE;
   instCmSepaClampTopUpDown.statDiagnostics.status := 16#7003;
   instCmSepaClampTopUpDown.statDiagnostics.subfunctionStatus := 16#0000;
   instCmSepaClampTopUpDown.statDiagnostics.stateNumber := 0;
   instCmSepaClampTopUpDown.statEnablePrevious := TRUE;
   instCmSepaClampTopUpDown.statFirstCall := FALSE;
   instCmSepaClampTopUpDown.statResetPrevious := FALSE;
   instCmSepaClampTopUpDown.statValid := TRUE;
   instCmSepaClampTopUpDown.statBusy := TRUE;
   instCmSepaClampTopUpDown.statError := FALSE;
   instCmSepaClampTopUpDown.statInterlockWorkOff := FALSE;
   instCmSepaClampTopUpDown.statInterlockHomeOff := FALSE;
   instCmSepaClampTopUpDown.statFbState := 50;
   instCmSepaClampTopUpDown.statFbStatePrevious := 50;
   instCmSepaClampTopUpDown.statErrorUserCleared := FALSE;
   instCmSepaClampTopUpDown.statErrorAutoCleared := FALSE;
   instCmSepaClampTopUpDown.statErrorState := 16#0000;
   instCmSepaClampTopUpDown.statDisablingCompleted := FALSE;
   instCmSepaClampTopUpDown.statFeedbackHomePos := FALSE;
   instCmSepaClampTopUpDown.statFeedbackWorkPos := TRUE;
   instCmSepaClampBottomUpDown.enable := TRUE;
   instCmSepaClampBottomUpDown.parentReferenceDesignator := WSTRING#'';
   instCmSepaClampBottomUpDown.feedbackHomePos := FALSE;
   instCmSepaClampBottomUpDown.feedbackWorkPos := TRUE;
   instCmSepaClampBottomUpDown.enableManualCmds := TRUE;
   instCmSepaClampBottomUpDown.interlockWorkPos := TRUE;
   instCmSepaClampBottomUpDown.interlockHomePos := FALSE;
   instCmSepaClampBottomUpDown.goToHomePos := FALSE;
   instCmSepaClampBottomUpDown.goToWorkPos := FALSE;
   instCmSepaClampBottomUpDown.statProcessValues.enable := TRUE;
   instCmSepaClampBottomUpDown.statProcessValues.referenceDesignator := WSTRING#'ClampBottomUpDown';
   instCmSepaClampBottomUpDown.statProcessValues.commandHomePos := FALSE;
   instCmSepaClampBottomUpDown.statProcessValues.commandWorkPos := FALSE;
   instCmSepaClampBottomUpDown.statProcessValues.goToHomePos := FALSE;
   instCmSepaClampBottomUpDown.statProcessValues.goToWorkPos := FALSE;
   instCmSepaClampBottomUpDown.statProcessValues.inHomePos := FALSE;
   instCmSepaClampBottomUpDown.statProcessValues.inWorkPos := TRUE;
   instCmSepaClampBottomUpDown.statProcessValues.reset := FALSE;
   instCmSepaClampBottomUpDown.statProcessValues.enableManualCmds := TRUE;
   instCmSepaClampBottomUpDown.statProcessValues.error := FALSE;
   instCmSepaClampBottomUpDown.statProcessValues.interlockHomePos := FALSE;
   instCmSepaClampBottomUpDown.statProcessValues.interlockWorkPos := TRUE;
   instCmSepaClampBottomUpDown.statProcessValues.status := 16#7102;
   instCmSepaClampBottomUpDown.statProcessValues.interlockWarningWorkPos := FALSE;
   instCmSepaClampBottomUpDown.statProcessValues.interlockWarningHomePos := FALSE;
   instCmSepaClampBottomUpDown.statCurrentInputs.commandHomePos := FALSE;
   instCmSepaClampBottomUpDown.statCurrentInputs.commandWorkPos := FALSE;
   instCmSepaClampBottomUpDown.statCurrentInputs.reset := FALSE;
   instCmSepaClampBottomUpDown.statPreviousInputs.commandHomePos := FALSE;
   instCmSepaClampBottomUpDown.statPreviousInputs.commandWorkPos := FALSE;
   instCmSepaClampBottomUpDown.statPreviousInputs.reset := FALSE;
   instCmSepaClampBottomUpDown.statCurrentInterface.commandHomePos := FALSE;
   instCmSepaClampBottomUpDown.statCurrentInterface.commandWorkPos := FALSE;
   instCmSepaClampBottomUpDown.statCurrentInterface.reset := FALSE;
   instCmSepaClampBottomUpDown.statPreviousInterface.commandHomePos := FALSE;
   instCmSepaClampBottomUpDown.statPreviousInterface.commandWorkPos := FALSE;
   instCmSepaClampBottomUpDown.statPreviousInterface.reset := FALSE;
   instCmSepaClampBottomUpDown.statEmptyDiagnostics.status := 16#0000;
   instCmSepaClampBottomUpDown.statEmptyDiagnostics.subfunctionStatus := 16#0000;
   instCmSepaClampBottomUpDown.statEmptyDiagnostics.stateNumber := 0;
   instCmSepaClampBottomUpDown.instTimerReachPos.PT := T#0MS;
   instCmSepaClampBottomUpDown.instTimerReachPos.IN := FALSE;
   instCmSepaClampBottomUpDown.instTimerLeavePos.PT := T#0MS;
   instCmSepaClampBottomUpDown.instTimerLeavePos.IN := FALSE;
   instCmSepaClampBottomUpDown.instTimerDiscrepancyCheck.PT := T#0MS;
   instCmSepaClampBottomUpDown.instTimerDiscrepancyCheck.IN := FALSE;
   instCmSepaClampBottomUpDown.statDisableAlarms := FALSE;
   instCmSepaClampBottomUpDown.statDiagnostics.status := 16#7003;
   instCmSepaClampBottomUpDown.statDiagnostics.subfunctionStatus := 16#0000;
   instCmSepaClampBottomUpDown.statDiagnostics.stateNumber := 0;
   instCmSepaClampBottomUpDown.statEnablePrevious := TRUE;
   instCmSepaClampBottomUpDown.statFirstCall := FALSE;
   instCmSepaClampBottomUpDown.statResetPrevious := FALSE;
   instCmSepaClampBottomUpDown.statValid := TRUE;
   instCmSepaClampBottomUpDown.statBusy := TRUE;
   instCmSepaClampBottomUpDown.statError := FALSE;
   instCmSepaClampBottomUpDown.statInterlockWorkOff := FALSE;
   instCmSepaClampBottomUpDown.statInterlockHomeOff := FALSE;
   instCmSepaClampBottomUpDown.statFbState := 50;
   instCmSepaClampBottomUpDown.statFbStatePrevious := 50;
   instCmSepaClampBottomUpDown.statErrorUserCleared := FALSE;
   instCmSepaClampBottomUpDown.statErrorAutoCleared := FALSE;
   instCmSepaClampBottomUpDown.statErrorState := 16#0000;
   instCmSepaClampBottomUpDown.statDisablingCompleted := FALSE;
   instCmSepaClampBottomUpDown.statFeedbackHomePos := FALSE;
   instCmSepaClampBottomUpDown.statFeedbackWorkPos := TRUE;
   instCmStackGripperOpenClose.enable := TRUE;
   instCmStackGripperOpenClose.parentReferenceDesignator := WSTRING#'';
   instCmStackGripperOpenClose.feedbackHomePos := FALSE;
   instCmStackGripperOpenClose.feedbackWorkPos := TRUE;
   instCmStackGripperOpenClose.enableManualCmds := TRUE;
   instCmStackGripperOpenClose.interlockWorkPos := TRUE;
   instCmStackGripperOpenClose.interlockHomePos := TRUE;
   instCmStackGripperOpenClose.goToHomePos := FALSE;
   instCmStackGripperOpenClose.goToWorkPos := FALSE;
   instCmStackGripperOpenClose.statProcessValues.enable := TRUE;
   instCmStackGripperOpenClose.statProcessValues.referenceDesignator := WSTRING#'GripperOpenClose';
   instCmStackGripperOpenClose.statProcessValues.commandHomePos := FALSE;
   instCmStackGripperOpenClose.statProcessValues.commandWorkPos := FALSE;
   instCmStackGripperOpenClose.statProcessValues.goToHomePos := FALSE;
   instCmStackGripperOpenClose.statProcessValues.goToWorkPos := FALSE;
   instCmStackGripperOpenClose.statProcessValues.inHomePos := FALSE;
   instCmStackGripperOpenClose.statProcessValues.inWorkPos := TRUE;
   instCmStackGripperOpenClose.statProcessValues.reset := FALSE;
   instCmStackGripperOpenClose.statProcessValues.enableManualCmds := TRUE;
   instCmStackGripperOpenClose.statProcessValues.error := FALSE;
   instCmStackGripperOpenClose.statProcessValues.interlockHomePos := TRUE;
   instCmStackGripperOpenClose.statProcessValues.interlockWorkPos := TRUE;
   instCmStackGripperOpenClose.statProcessValues.status := 16#7003;
   instCmStackGripperOpenClose.statProcessValues.interlockWarningWorkPos := FALSE;
   instCmStackGripperOpenClose.statProcessValues.interlockWarningHomePos := FALSE;
   instCmStackGripperOpenClose.statCurrentInputs.commandHomePos := FALSE;
   instCmStackGripperOpenClose.statCurrentInputs.commandWorkPos := FALSE;
   instCmStackGripperOpenClose.statCurrentInputs.reset := FALSE;
   instCmStackGripperOpenClose.statPreviousInputs.commandHomePos := FALSE;
   instCmStackGripperOpenClose.statPreviousInputs.commandWorkPos := FALSE;
   instCmStackGripperOpenClose.statPreviousInputs.reset := FALSE;
   instCmStackGripperOpenClose.statCurrentInterface.commandHomePos := FALSE;
   instCmStackGripperOpenClose.statCurrentInterface.commandWorkPos := FALSE;
   instCmStackGripperOpenClose.statCurrentInterface.reset := FALSE;
   instCmStackGripperOpenClose.statPreviousInterface.commandHomePos := FALSE;
   instCmStackGripperOpenClose.statPreviousInterface.commandWorkPos := FALSE;
   instCmStackGripperOpenClose.statPreviousInterface.reset := FALSE;
   instCmStackGripperOpenClose.statEmptyDiagnostics.status := 16#0000;
   instCmStackGripperOpenClose.statEmptyDiagnostics.subfunctionStatus := 16#0000;
   instCmStackGripperOpenClose.statEmptyDiagnostics.stateNumber := 0;
   instCmStackGripperOpenClose.instTimerReachPos.PT := T#0MS;
   instCmStackGripperOpenClose.instTimerReachPos.IN := FALSE;
   instCmStackGripperOpenClose.instTimerLeavePos.PT := T#0MS;
   instCmStackGripperOpenClose.instTimerLeavePos.IN := FALSE;
   instCmStackGripperOpenClose.instTimerDiscrepancyCheck.PT := T#0MS;
   instCmStackGripperOpenClose.instTimerDiscrepancyCheck.IN := FALSE;
   instCmStackGripperOpenClose.statDisableAlarms := FALSE;
   instCmStackGripperOpenClose.statDiagnostics.status := 16#7003;
   instCmStackGripperOpenClose.statDiagnostics.subfunctionStatus := 16#0000;
   instCmStackGripperOpenClose.statDiagnostics.stateNumber := 0;
   instCmStackGripperOpenClose.statEnablePrevious := TRUE;
   instCmStackGripperOpenClose.statFirstCall := FALSE;
   instCmStackGripperOpenClose.statResetPrevious := FALSE;
   instCmStackGripperOpenClose.statValid := TRUE;
   instCmStackGripperOpenClose.statBusy := TRUE;
   instCmStackGripperOpenClose.statError := FALSE;
   instCmStackGripperOpenClose.statInterlockWorkOff := FALSE;
   instCmStackGripperOpenClose.statInterlockHomeOff := FALSE;
   instCmStackGripperOpenClose.statFbState := 50;
   instCmStackGripperOpenClose.statFbStatePrevious := 50;
   instCmStackGripperOpenClose.statErrorUserCleared := FALSE;
   instCmStackGripperOpenClose.statErrorAutoCleared := FALSE;
   instCmStackGripperOpenClose.statErrorState := 16#0000;
   instCmStackGripperOpenClose.statDisablingCompleted := FALSE;
   instCmStackGripperOpenClose.statFeedbackHomePos := FALSE;
   instCmStackGripperOpenClose.statFeedbackWorkPos := TRUE;
   instCmStackGripperFwdBwd.enable := TRUE;
   instCmStackGripperFwdBwd.parentReferenceDesignator := WSTRING#'';
   instCmStackGripperFwdBwd.feedbackHomePos := FALSE;
   instCmStackGripperFwdBwd.feedbackWorkPos := FALSE;
   instCmStackGripperFwdBwd.enableManualCmds := TRUE;
   instCmStackGripperFwdBwd.interlockWorkPos := FALSE;
   instCmStackGripperFwdBwd.interlockHomePos := TRUE;
   instCmStackGripperFwdBwd.goToHomePos := FALSE;
   instCmStackGripperFwdBwd.goToWorkPos := FALSE;
   instCmStackGripperFwdBwd.statProcessValues.enable := TRUE;
   instCmStackGripperFwdBwd.statProcessValues.referenceDesignator := WSTRING#'GripperFwdBwd';
   instCmStackGripperFwdBwd.statProcessValues.commandHomePos := FALSE;
   instCmStackGripperFwdBwd.statProcessValues.commandWorkPos := FALSE;
   instCmStackGripperFwdBwd.statProcessValues.goToHomePos := FALSE;
   instCmStackGripperFwdBwd.statProcessValues.goToWorkPos := FALSE;
   instCmStackGripperFwdBwd.statProcessValues.inHomePos := FALSE;
   instCmStackGripperFwdBwd.statProcessValues.inWorkPos := FALSE;
   instCmStackGripperFwdBwd.statProcessValues.reset := FALSE;
   instCmStackGripperFwdBwd.statProcessValues.enableManualCmds := TRUE;
   instCmStackGripperFwdBwd.statProcessValues.error := FALSE;
   instCmStackGripperFwdBwd.statProcessValues.interlockHomePos := TRUE;
   instCmStackGripperFwdBwd.statProcessValues.interlockWorkPos := FALSE;
   instCmStackGripperFwdBwd.statProcessValues.status := 16#7101;
   instCmStackGripperFwdBwd.statProcessValues.interlockWarningWorkPos := FALSE;
   instCmStackGripperFwdBwd.statProcessValues.interlockWarningHomePos := FALSE;
   instCmStackGripperFwdBwd.statCurrentInputs.commandHomePos := FALSE;
   instCmStackGripperFwdBwd.statCurrentInputs.commandWorkPos := FALSE;
   instCmStackGripperFwdBwd.statCurrentInputs.reset := FALSE;
   instCmStackGripperFwdBwd.statPreviousInputs.commandHomePos := FALSE;
   instCmStackGripperFwdBwd.statPreviousInputs.commandWorkPos := FALSE;
   instCmStackGripperFwdBwd.statPreviousInputs.reset := FALSE;
   instCmStackGripperFwdBwd.statCurrentInterface.commandHomePos := FALSE;
   instCmStackGripperFwdBwd.statCurrentInterface.commandWorkPos := FALSE;
   instCmStackGripperFwdBwd.statCurrentInterface.reset := FALSE;
   instCmStackGripperFwdBwd.statPreviousInterface.commandHomePos := FALSE;
   instCmStackGripperFwdBwd.statPreviousInterface.commandWorkPos := FALSE;
   instCmStackGripperFwdBwd.statPreviousInterface.reset := FALSE;
   instCmStackGripperFwdBwd.statEmptyDiagnostics.status := 16#0000;
   instCmStackGripperFwdBwd.statEmptyDiagnostics.subfunctionStatus := 16#0000;
   instCmStackGripperFwdBwd.statEmptyDiagnostics.stateNumber := 0;
   instCmStackGripperFwdBwd.instTimerReachPos.PT := T#0MS;
   instCmStackGripperFwdBwd.instTimerReachPos.IN := FALSE;
   instCmStackGripperFwdBwd.instTimerLeavePos.PT := T#0MS;
   instCmStackGripperFwdBwd.instTimerLeavePos.IN := FALSE;
   instCmStackGripperFwdBwd.instTimerDiscrepancyCheck.PT := T#0MS;
   instCmStackGripperFwdBwd.instTimerDiscrepancyCheck.IN := FALSE;
   instCmStackGripperFwdBwd.statDisableAlarms := FALSE;
   instCmStackGripperFwdBwd.statDiagnostics.status := 16#7003;
   instCmStackGripperFwdBwd.statDiagnostics.subfunctionStatus := 16#0000;
   instCmStackGripperFwdBwd.statDiagnostics.stateNumber := 0;
   instCmStackGripperFwdBwd.statEnablePrevious := TRUE;
   instCmStackGripperFwdBwd.statFirstCall := FALSE;
   instCmStackGripperFwdBwd.statResetPrevious := FALSE;
   instCmStackGripperFwdBwd.statValid := TRUE;
   instCmStackGripperFwdBwd.statBusy := TRUE;
   instCmStackGripperFwdBwd.statError := FALSE;
   instCmStackGripperFwdBwd.statInterlockWorkOff := FALSE;
   instCmStackGripperFwdBwd.statInterlockHomeOff := FALSE;
   instCmStackGripperFwdBwd.statFbState := 50;
   instCmStackGripperFwdBwd.statFbStatePrevious := 50;
   instCmStackGripperFwdBwd.statErrorUserCleared := FALSE;
   instCmStackGripperFwdBwd.statErrorAutoCleared := FALSE;
   instCmStackGripperFwdBwd.statErrorState := 16#0000;
   instCmStackGripperFwdBwd.statDisablingCompleted := FALSE;
   instCmStackGripperFwdBwd.statFeedbackHomePos := FALSE;
   instCmStackGripperFwdBwd.statFeedbackWorkPos := FALSE;
   instCmJRWinderClampTopRearUpDown.enable := TRUE;
   instCmJRWinderClampTopRearUpDown.parentReferenceDesignator := WSTRING#'';
   instCmJRWinderClampTopRearUpDown.feedbackHomePos := FALSE;
   instCmJRWinderClampTopRearUpDown.feedbackWorkPos := FALSE;
   instCmJRWinderClampTopRearUpDown.enableManualCmds := TRUE;
   instCmJRWinderClampTopRearUpDown.interlockWorkPos := TRUE;
   instCmJRWinderClampTopRearUpDown.interlockHomePos := TRUE;
   instCmJRWinderClampTopRearUpDown.goToHomePos := FALSE;
   instCmJRWinderClampTopRearUpDown.goToWorkPos := FALSE;
   instCmJRWinderClampTopRearUpDown.statProcessValues.enable := TRUE;
   instCmJRWinderClampTopRearUpDown.statProcessValues.referenceDesignator := WSTRING#'JRClampTopRearUpDown.';
   instCmJRWinderClampTopRearUpDown.statProcessValues.commandHomePos := FALSE;
   instCmJRWinderClampTopRearUpDown.statProcessValues.commandWorkPos := FALSE;
   instCmJRWinderClampTopRearUpDown.statProcessValues.goToHomePos := FALSE;
   instCmJRWinderClampTopRearUpDown.statProcessValues.goToWorkPos := FALSE;
   instCmJRWinderClampTopRearUpDown.statProcessValues.inHomePos := FALSE;
   instCmJRWinderClampTopRearUpDown.statProcessValues.inWorkPos := FALSE;
   instCmJRWinderClampTopRearUpDown.statProcessValues.reset := FALSE;
   instCmJRWinderClampTopRearUpDown.statProcessValues.enableManualCmds := TRUE;
   instCmJRWinderClampTopRearUpDown.statProcessValues.error := FALSE;
   instCmJRWinderClampTopRearUpDown.statProcessValues.interlockHomePos := TRUE;
   instCmJRWinderClampTopRearUpDown.statProcessValues.interlockWorkPos := TRUE;
   instCmJRWinderClampTopRearUpDown.statProcessValues.status := 16#7003;
   instCmJRWinderClampTopRearUpDown.statProcessValues.interlockWarningWorkPos := FALSE;
   instCmJRWinderClampTopRearUpDown.statProcessValues.interlockWarningHomePos := FALSE;
   instCmJRWinderClampTopRearUpDown.statCurrentInputs.commandHomePos := FALSE;
   instCmJRWinderClampTopRearUpDown.statCurrentInputs.commandWorkPos := FALSE;
   instCmJRWinderClampTopRearUpDown.statCurrentInputs.reset := FALSE;
   instCmJRWinderClampTopRearUpDown.statPreviousInputs.commandHomePos := FALSE;
   instCmJRWinderClampTopRearUpDown.statPreviousInputs.commandWorkPos := FALSE;
   instCmJRWinderClampTopRearUpDown.statPreviousInputs.reset := FALSE;
   instCmJRWinderClampTopRearUpDown.statCurrentInterface.commandHomePos := FALSE;
   instCmJRWinderClampTopRearUpDown.statCurrentInterface.commandWorkPos := FALSE;
   instCmJRWinderClampTopRearUpDown.statCurrentInterface.reset := FALSE;
   instCmJRWinderClampTopRearUpDown.statPreviousInterface.commandHomePos := FALSE;
   instCmJRWinderClampTopRearUpDown.statPreviousInterface.commandWorkPos := FALSE;
   instCmJRWinderClampTopRearUpDown.statPreviousInterface.reset := FALSE;
   instCmJRWinderClampTopRearUpDown.statEmptyDiagnostics.status := 16#0000;
   instCmJRWinderClampTopRearUpDown.statEmptyDiagnostics.subfunctionStatus := 16#0000;
   instCmJRWinderClampTopRearUpDown.statEmptyDiagnostics.stateNumber := 0;
   instCmJRWinderClampTopRearUpDown.instTimerReachPos.PT := T#0MS;
   instCmJRWinderClampTopRearUpDown.instTimerReachPos.IN := FALSE;
   instCmJRWinderClampTopRearUpDown.instTimerLeavePos.PT := T#0MS;
   instCmJRWinderClampTopRearUpDown.instTimerLeavePos.IN := FALSE;
   instCmJRWinderClampTopRearUpDown.instTimerDiscrepancyCheck.PT := T#0MS;
   instCmJRWinderClampTopRearUpDown.instTimerDiscrepancyCheck.IN := FALSE;
   instCmJRWinderClampTopRearUpDown.statDisableAlarms := FALSE;
   instCmJRWinderClampTopRearUpDown.statDiagnostics.status := 16#7003;
   instCmJRWinderClampTopRearUpDown.statDiagnostics.subfunctionStatus := 16#0000;
   instCmJRWinderClampTopRearUpDown.statDiagnostics.stateNumber := 0;
   instCmJRWinderClampTopRearUpDown.statEnablePrevious := TRUE;
   instCmJRWinderClampTopRearUpDown.statFirstCall := FALSE;
   instCmJRWinderClampTopRearUpDown.statResetPrevious := FALSE;
   instCmJRWinderClampTopRearUpDown.statValid := TRUE;
   instCmJRWinderClampTopRearUpDown.statBusy := TRUE;
   instCmJRWinderClampTopRearUpDown.statError := FALSE;
   instCmJRWinderClampTopRearUpDown.statInterlockWorkOff := FALSE;
   instCmJRWinderClampTopRearUpDown.statInterlockHomeOff := FALSE;
   instCmJRWinderClampTopRearUpDown.statFbState := 50;
   instCmJRWinderClampTopRearUpDown.statFbStatePrevious := 50;
   instCmJRWinderClampTopRearUpDown.statErrorUserCleared := FALSE;
   instCmJRWinderClampTopRearUpDown.statErrorAutoCleared := FALSE;
   instCmJRWinderClampTopRearUpDown.statErrorState := 16#0000;
   instCmJRWinderClampTopRearUpDown.statDisablingCompleted := FALSE;
   instCmJRWinderClampTopRearUpDown.statFeedbackHomePos := FALSE;
   instCmJRWinderClampTopRearUpDown.statFeedbackWorkPos := FALSE;
   instCmJRWinderClampBtmRearUpDown.enable := TRUE;
   instCmJRWinderClampBtmRearUpDown.parentReferenceDesignator := WSTRING#'';
   instCmJRWinderClampBtmRearUpDown.feedbackHomePos := FALSE;
   instCmJRWinderClampBtmRearUpDown.feedbackWorkPos := FALSE;
   instCmJRWinderClampBtmRearUpDown.enableManualCmds := TRUE;
   instCmJRWinderClampBtmRearUpDown.interlockWorkPos := TRUE;
   instCmJRWinderClampBtmRearUpDown.interlockHomePos := TRUE;
   instCmJRWinderClampBtmRearUpDown.goToHomePos := FALSE;
   instCmJRWinderClampBtmRearUpDown.goToWorkPos := FALSE;
   instCmJRWinderClampBtmRearUpDown.statProcessValues.enable := TRUE;
   instCmJRWinderClampBtmRearUpDown.statProcessValues.referenceDesignator := WSTRING#'JRClampBtmRearUpDown.';
   instCmJRWinderClampBtmRearUpDown.statProcessValues.commandHomePos := FALSE;
   instCmJRWinderClampBtmRearUpDown.statProcessValues.commandWorkPos := FALSE;
   instCmJRWinderClampBtmRearUpDown.statProcessValues.goToHomePos := FALSE;
   instCmJRWinderClampBtmRearUpDown.statProcessValues.goToWorkPos := FALSE;
   instCmJRWinderClampBtmRearUpDown.statProcessValues.inHomePos := FALSE;
   instCmJRWinderClampBtmRearUpDown.statProcessValues.inWorkPos := FALSE;
   instCmJRWinderClampBtmRearUpDown.statProcessValues.reset := FALSE;
   instCmJRWinderClampBtmRearUpDown.statProcessValues.enableManualCmds := TRUE;
   instCmJRWinderClampBtmRearUpDown.statProcessValues.error := FALSE;
   instCmJRWinderClampBtmRearUpDown.statProcessValues.interlockHomePos := TRUE;
   instCmJRWinderClampBtmRearUpDown.statProcessValues.interlockWorkPos := TRUE;
   instCmJRWinderClampBtmRearUpDown.statProcessValues.status := 16#7003;
   instCmJRWinderClampBtmRearUpDown.statProcessValues.interlockWarningWorkPos := FALSE;
   instCmJRWinderClampBtmRearUpDown.statProcessValues.interlockWarningHomePos := FALSE;
   instCmJRWinderClampBtmRearUpDown.statCurrentInputs.commandHomePos := FALSE;
   instCmJRWinderClampBtmRearUpDown.statCurrentInputs.commandWorkPos := FALSE;
   instCmJRWinderClampBtmRearUpDown.statCurrentInputs.reset := FALSE;
   instCmJRWinderClampBtmRearUpDown.statPreviousInputs.commandHomePos := FALSE;
   instCmJRWinderClampBtmRearUpDown.statPreviousInputs.commandWorkPos := FALSE;
   instCmJRWinderClampBtmRearUpDown.statPreviousInputs.reset := FALSE;
   instCmJRWinderClampBtmRearUpDown.statCurrentInterface.commandHomePos := FALSE;
   instCmJRWinderClampBtmRearUpDown.statCurrentInterface.commandWorkPos := FALSE;
   instCmJRWinderClampBtmRearUpDown.statCurrentInterface.reset := FALSE;
   instCmJRWinderClampBtmRearUpDown.statPreviousInterface.commandHomePos := FALSE;
   instCmJRWinderClampBtmRearUpDown.statPreviousInterface.commandWorkPos := FALSE;
   instCmJRWinderClampBtmRearUpDown.statPreviousInterface.reset := FALSE;
   instCmJRWinderClampBtmRearUpDown.statEmptyDiagnostics.status := 16#0000;
   instCmJRWinderClampBtmRearUpDown.statEmptyDiagnostics.subfunctionStatus := 16#0000;
   instCmJRWinderClampBtmRearUpDown.statEmptyDiagnostics.stateNumber := 0;
   instCmJRWinderClampBtmRearUpDown.instTimerReachPos.PT := T#0MS;
   instCmJRWinderClampBtmRearUpDown.instTimerReachPos.IN := FALSE;
   instCmJRWinderClampBtmRearUpDown.instTimerLeavePos.PT := T#0MS;
   instCmJRWinderClampBtmRearUpDown.instTimerLeavePos.IN := FALSE;
   instCmJRWinderClampBtmRearUpDown.instTimerDiscrepancyCheck.PT := T#0MS;
   instCmJRWinderClampBtmRearUpDown.instTimerDiscrepancyCheck.IN := FALSE;
   instCmJRWinderClampBtmRearUpDown.statDisableAlarms := FALSE;
   instCmJRWinderClampBtmRearUpDown.statDiagnostics.status := 16#7003;
   instCmJRWinderClampBtmRearUpDown.statDiagnostics.subfunctionStatus := 16#0000;
   instCmJRWinderClampBtmRearUpDown.statDiagnostics.stateNumber := 0;
   instCmJRWinderClampBtmRearUpDown.statEnablePrevious := TRUE;
   instCmJRWinderClampBtmRearUpDown.statFirstCall := FALSE;
   instCmJRWinderClampBtmRearUpDown.statResetPrevious := FALSE;
   instCmJRWinderClampBtmRearUpDown.statValid := TRUE;
   instCmJRWinderClampBtmRearUpDown.statBusy := TRUE;
   instCmJRWinderClampBtmRearUpDown.statError := FALSE;
   instCmJRWinderClampBtmRearUpDown.statInterlockWorkOff := FALSE;
   instCmJRWinderClampBtmRearUpDown.statInterlockHomeOff := FALSE;
   instCmJRWinderClampBtmRearUpDown.statFbState := 50;
   instCmJRWinderClampBtmRearUpDown.statFbStatePrevious := 50;
   instCmJRWinderClampBtmRearUpDown.statErrorUserCleared := FALSE;
   instCmJRWinderClampBtmRearUpDown.statErrorAutoCleared := FALSE;
   instCmJRWinderClampBtmRearUpDown.statErrorState := 16#0000;
   instCmJRWinderClampBtmRearUpDown.statDisablingCompleted := FALSE;
   instCmJRWinderClampBtmRearUpDown.statFeedbackHomePos := FALSE;
   instCmJRWinderClampBtmRearUpDown.statFeedbackWorkPos := FALSE;
   instCmJRWinderClampTopFrontUpDown.enable := TRUE;
   instCmJRWinderClampTopFrontUpDown.parentReferenceDesignator := WSTRING#'';
   instCmJRWinderClampTopFrontUpDown.feedbackHomePos := FALSE;
   instCmJRWinderClampTopFrontUpDown.feedbackWorkPos := FALSE;
   instCmJRWinderClampTopFrontUpDown.enableManualCmds := TRUE;
   instCmJRWinderClampTopFrontUpDown.interlockWorkPos := TRUE;
   instCmJRWinderClampTopFrontUpDown.interlockHomePos := TRUE;
   instCmJRWinderClampTopFrontUpDown.goToHomePos := FALSE;
   instCmJRWinderClampTopFrontUpDown.goToWorkPos := FALSE;
   instCmJRWinderClampTopFrontUpDown.statProcessValues.enable := TRUE;
   instCmJRWinderClampTopFrontUpDown.statProcessValues.referenceDesignator := WSTRING#'JRClampTopFrontUpDown.';
   instCmJRWinderClampTopFrontUpDown.statProcessValues.commandHomePos := FALSE;
   instCmJRWinderClampTopFrontUpDown.statProcessValues.commandWorkPos := FALSE;
   instCmJRWinderClampTopFrontUpDown.statProcessValues.goToHomePos := FALSE;
   instCmJRWinderClampTopFrontUpDown.statProcessValues.goToWorkPos := FALSE;
   instCmJRWinderClampTopFrontUpDown.statProcessValues.inHomePos := FALSE;
   instCmJRWinderClampTopFrontUpDown.statProcessValues.inWorkPos := FALSE;
   instCmJRWinderClampTopFrontUpDown.statProcessValues.reset := FALSE;
   instCmJRWinderClampTopFrontUpDown.statProcessValues.enableManualCmds := TRUE;
   instCmJRWinderClampTopFrontUpDown.statProcessValues.error := FALSE;
   instCmJRWinderClampTopFrontUpDown.statProcessValues.interlockHomePos := TRUE;
   instCmJRWinderClampTopFrontUpDown.statProcessValues.interlockWorkPos := TRUE;
   instCmJRWinderClampTopFrontUpDown.statProcessValues.status := 16#7003;
   instCmJRWinderClampTopFrontUpDown.statProcessValues.interlockWarningWorkPos := FALSE;
   instCmJRWinderClampTopFrontUpDown.statProcessValues.interlockWarningHomePos := FALSE;
   instCmJRWinderClampTopFrontUpDown.statCurrentInputs.commandHomePos := FALSE;
   instCmJRWinderClampTopFrontUpDown.statCurrentInputs.commandWorkPos := FALSE;
   instCmJRWinderClampTopFrontUpDown.statCurrentInputs.reset := FALSE;
   instCmJRWinderClampTopFrontUpDown.statPreviousInputs.commandHomePos := FALSE;
   instCmJRWinderClampTopFrontUpDown.statPreviousInputs.commandWorkPos := FALSE;
   instCmJRWinderClampTopFrontUpDown.statPreviousInputs.reset := FALSE;
   instCmJRWinderClampTopFrontUpDown.statCurrentInterface.commandHomePos := FALSE;
   instCmJRWinderClampTopFrontUpDown.statCurrentInterface.commandWorkPos := FALSE;
   instCmJRWinderClampTopFrontUpDown.statCurrentInterface.reset := FALSE;
   instCmJRWinderClampTopFrontUpDown.statPreviousInterface.commandHomePos := FALSE;
   instCmJRWinderClampTopFrontUpDown.statPreviousInterface.commandWorkPos := FALSE;
   instCmJRWinderClampTopFrontUpDown.statPreviousInterface.reset := FALSE;
   instCmJRWinderClampTopFrontUpDown.statEmptyDiagnostics.status := 16#0000;
   instCmJRWinderClampTopFrontUpDown.statEmptyDiagnostics.subfunctionStatus := 16#0000;
   instCmJRWinderClampTopFrontUpDown.statEmptyDiagnostics.stateNumber := 0;
   instCmJRWinderClampTopFrontUpDown.instTimerReachPos.PT := T#0MS;
   instCmJRWinderClampTopFrontUpDown.instTimerReachPos.IN := FALSE;
   instCmJRWinderClampTopFrontUpDown.instTimerLeavePos.PT := T#0MS;
   instCmJRWinderClampTopFrontUpDown.instTimerLeavePos.IN := FALSE;
   instCmJRWinderClampTopFrontUpDown.instTimerDiscrepancyCheck.PT := T#0MS;
   instCmJRWinderClampTopFrontUpDown.instTimerDiscrepancyCheck.IN := FALSE;
   instCmJRWinderClampTopFrontUpDown.statDisableAlarms := FALSE;
   instCmJRWinderClampTopFrontUpDown.statDiagnostics.status := 16#7003;
   instCmJRWinderClampTopFrontUpDown.statDiagnostics.subfunctionStatus := 16#0000;
   instCmJRWinderClampTopFrontUpDown.statDiagnostics.stateNumber := 0;
   instCmJRWinderClampTopFrontUpDown.statEnablePrevious := TRUE;
   instCmJRWinderClampTopFrontUpDown.statFirstCall := FALSE;
   instCmJRWinderClampTopFrontUpDown.statResetPrevious := FALSE;
   instCmJRWinderClampTopFrontUpDown.statValid := TRUE;
   instCmJRWinderClampTopFrontUpDown.statBusy := TRUE;
   instCmJRWinderClampTopFrontUpDown.statError := FALSE;
   instCmJRWinderClampTopFrontUpDown.statInterlockWorkOff := FALSE;
   instCmJRWinderClampTopFrontUpDown.statInterlockHomeOff := FALSE;
   instCmJRWinderClampTopFrontUpDown.statFbState := 50;
   instCmJRWinderClampTopFrontUpDown.statFbStatePrevious := 50;
   instCmJRWinderClampTopFrontUpDown.statErrorUserCleared := FALSE;
   instCmJRWinderClampTopFrontUpDown.statErrorAutoCleared := FALSE;
   instCmJRWinderClampTopFrontUpDown.statErrorState := 16#0000;
   instCmJRWinderClampTopFrontUpDown.statDisablingCompleted := FALSE;
   instCmJRWinderClampTopFrontUpDown.statFeedbackHomePos := FALSE;
   instCmJRWinderClampTopFrontUpDown.statFeedbackWorkPos := FALSE;
   instCmJRWinderClampBtmFrontUpDown.enable := TRUE;
   instCmJRWinderClampBtmFrontUpDown.parentReferenceDesignator := WSTRING#'';
   instCmJRWinderClampBtmFrontUpDown.feedbackHomePos := FALSE;
   instCmJRWinderClampBtmFrontUpDown.feedbackWorkPos := FALSE;
   instCmJRWinderClampBtmFrontUpDown.enableManualCmds := TRUE;
   instCmJRWinderClampBtmFrontUpDown.interlockWorkPos := TRUE;
   instCmJRWinderClampBtmFrontUpDown.interlockHomePos := TRUE;
   instCmJRWinderClampBtmFrontUpDown.goToHomePos := FALSE;
   instCmJRWinderClampBtmFrontUpDown.goToWorkPos := FALSE;
   instCmJRWinderClampBtmFrontUpDown.statProcessValues.enable := TRUE;
   instCmJRWinderClampBtmFrontUpDown.statProcessValues.referenceDesignator := WSTRING#'JRClampBtmFrontUpDown.';
   instCmJRWinderClampBtmFrontUpDown.statProcessValues.commandHomePos := FALSE;
   instCmJRWinderClampBtmFrontUpDown.statProcessValues.commandWorkPos := FALSE;
   instCmJRWinderClampBtmFrontUpDown.statProcessValues.goToHomePos := FALSE;
   instCmJRWinderClampBtmFrontUpDown.statProcessValues.goToWorkPos := FALSE;
   instCmJRWinderClampBtmFrontUpDown.statProcessValues.inHomePos := FALSE;
   instCmJRWinderClampBtmFrontUpDown.statProcessValues.inWorkPos := FALSE;
   instCmJRWinderClampBtmFrontUpDown.statProcessValues.reset := FALSE;
   instCmJRWinderClampBtmFrontUpDown.statProcessValues.enableManualCmds := TRUE;
   instCmJRWinderClampBtmFrontUpDown.statProcessValues.error := FALSE;
   instCmJRWinderClampBtmFrontUpDown.statProcessValues.interlockHomePos := TRUE;
   instCmJRWinderClampBtmFrontUpDown.statProcessValues.interlockWorkPos := TRUE;
   instCmJRWinderClampBtmFrontUpDown.statProcessValues.status := 16#7003;
   instCmJRWinderClampBtmFrontUpDown.statProcessValues.interlockWarningWorkPos := FALSE;
   instCmJRWinderClampBtmFrontUpDown.statProcessValues.interlockWarningHomePos := FALSE;
   instCmJRWinderClampBtmFrontUpDown.statCurrentInputs.commandHomePos := FALSE;
   instCmJRWinderClampBtmFrontUpDown.statCurrentInputs.commandWorkPos := FALSE;
   instCmJRWinderClampBtmFrontUpDown.statCurrentInputs.reset := FALSE;
   instCmJRWinderClampBtmFrontUpDown.statPreviousInputs.commandHomePos := FALSE;
   instCmJRWinderClampBtmFrontUpDown.statPreviousInputs.commandWorkPos := FALSE;
   instCmJRWinderClampBtmFrontUpDown.statPreviousInputs.reset := FALSE;
   instCmJRWinderClampBtmFrontUpDown.statCurrentInterface.commandHomePos := FALSE;
   instCmJRWinderClampBtmFrontUpDown.statCurrentInterface.commandWorkPos := FALSE;
   instCmJRWinderClampBtmFrontUpDown.statCurrentInterface.reset := FALSE;
   instCmJRWinderClampBtmFrontUpDown.statPreviousInterface.commandHomePos := FALSE;
   instCmJRWinderClampBtmFrontUpDown.statPreviousInterface.commandWorkPos := FALSE;
   instCmJRWinderClampBtmFrontUpDown.statPreviousInterface.reset := FALSE;
   instCmJRWinderClampBtmFrontUpDown.statEmptyDiagnostics.status := 16#0000;
   instCmJRWinderClampBtmFrontUpDown.statEmptyDiagnostics.subfunctionStatus := 16#0000;
   instCmJRWinderClampBtmFrontUpDown.statEmptyDiagnostics.stateNumber := 0;
   instCmJRWinderClampBtmFrontUpDown.instTimerReachPos.PT := T#0MS;
   instCmJRWinderClampBtmFrontUpDown.instTimerReachPos.IN := FALSE;
   instCmJRWinderClampBtmFrontUpDown.instTimerLeavePos.PT := T#0MS;
   instCmJRWinderClampBtmFrontUpDown.instTimerLeavePos.IN := FALSE;
   instCmJRWinderClampBtmFrontUpDown.instTimerDiscrepancyCheck.PT := T#0MS;
   instCmJRWinderClampBtmFrontUpDown.instTimerDiscrepancyCheck.IN := FALSE;
   instCmJRWinderClampBtmFrontUpDown.statDisableAlarms := FALSE;
   instCmJRWinderClampBtmFrontUpDown.statDiagnostics.status := 16#7003;
   instCmJRWinderClampBtmFrontUpDown.statDiagnostics.subfunctionStatus := 16#0000;
   instCmJRWinderClampBtmFrontUpDown.statDiagnostics.stateNumber := 0;
   instCmJRWinderClampBtmFrontUpDown.statEnablePrevious := TRUE;
   instCmJRWinderClampBtmFrontUpDown.statFirstCall := FALSE;
   instCmJRWinderClampBtmFrontUpDown.statResetPrevious := FALSE;
   instCmJRWinderClampBtmFrontUpDown.statValid := TRUE;
   instCmJRWinderClampBtmFrontUpDown.statBusy := TRUE;
   instCmJRWinderClampBtmFrontUpDown.statError := FALSE;
   instCmJRWinderClampBtmFrontUpDown.statInterlockWorkOff := FALSE;
   instCmJRWinderClampBtmFrontUpDown.statInterlockHomeOff := FALSE;
   instCmJRWinderClampBtmFrontUpDown.statFbState := 50;
   instCmJRWinderClampBtmFrontUpDown.statFbStatePrevious := 50;
   instCmJRWinderClampBtmFrontUpDown.statErrorUserCleared := FALSE;
   instCmJRWinderClampBtmFrontUpDown.statErrorAutoCleared := FALSE;
   instCmJRWinderClampBtmFrontUpDown.statErrorState := 16#0000;
   instCmJRWinderClampBtmFrontUpDown.statDisablingCompleted := FALSE;
   instCmJRWinderClampBtmFrontUpDown.statFeedbackHomePos := FALSE;
   instCmJRWinderClampBtmFrontUpDown.statFeedbackWorkPos := FALSE;
   instCmPusherRollerFwdBwd.enable := TRUE;
   instCmPusherRollerFwdBwd.parentReferenceDesignator := WSTRING#'';
   instCmPusherRollerFwdBwd.feedbackHomePos := FALSE;
   instCmPusherRollerFwdBwd.feedbackWorkPos := FALSE;
   instCmPusherRollerFwdBwd.enableManualCmds := TRUE;
   instCmPusherRollerFwdBwd.interlockWorkPos := FALSE;
   instCmPusherRollerFwdBwd.interlockHomePos := FALSE;
   instCmPusherRollerFwdBwd.goToHomePos := FALSE;
   instCmPusherRollerFwdBwd.goToWorkPos := FALSE;
   instCmPusherRollerFwdBwd.statProcessValues.enable := TRUE;
   instCmPusherRollerFwdBwd.statProcessValues.referenceDesignator := WSTRING#'PusherRollerFwdBwd';
   instCmPusherRollerFwdBwd.statProcessValues.commandHomePos := FALSE;
   instCmPusherRollerFwdBwd.statProcessValues.commandWorkPos := FALSE;
   instCmPusherRollerFwdBwd.statProcessValues.goToHomePos := FALSE;
   instCmPusherRollerFwdBwd.statProcessValues.goToWorkPos := FALSE;
   instCmPusherRollerFwdBwd.statProcessValues.inHomePos := FALSE;
   instCmPusherRollerFwdBwd.statProcessValues.inWorkPos := FALSE;
   instCmPusherRollerFwdBwd.statProcessValues.reset := FALSE;
   instCmPusherRollerFwdBwd.statProcessValues.enableManualCmds := TRUE;
   instCmPusherRollerFwdBwd.statProcessValues.error := FALSE;
   instCmPusherRollerFwdBwd.statProcessValues.interlockHomePos := FALSE;
   instCmPusherRollerFwdBwd.statProcessValues.interlockWorkPos := FALSE;
   instCmPusherRollerFwdBwd.statProcessValues.status := 16#7100;
   instCmPusherRollerFwdBwd.statProcessValues.interlockWarningWorkPos := FALSE;
   instCmPusherRollerFwdBwd.statProcessValues.interlockWarningHomePos := FALSE;
   instCmPusherRollerFwdBwd.statCurrentInputs.commandHomePos := FALSE;
   instCmPusherRollerFwdBwd.statCurrentInputs.commandWorkPos := FALSE;
   instCmPusherRollerFwdBwd.statCurrentInputs.reset := FALSE;
   instCmPusherRollerFwdBwd.statPreviousInputs.commandHomePos := FALSE;
   instCmPusherRollerFwdBwd.statPreviousInputs.commandWorkPos := FALSE;
   instCmPusherRollerFwdBwd.statPreviousInputs.reset := FALSE;
   instCmPusherRollerFwdBwd.statCurrentInterface.commandHomePos := FALSE;
   instCmPusherRollerFwdBwd.statCurrentInterface.commandWorkPos := FALSE;
   instCmPusherRollerFwdBwd.statCurrentInterface.reset := FALSE;
   instCmPusherRollerFwdBwd.statPreviousInterface.commandHomePos := FALSE;
   instCmPusherRollerFwdBwd.statPreviousInterface.commandWorkPos := FALSE;
   instCmPusherRollerFwdBwd.statPreviousInterface.reset := FALSE;
   instCmPusherRollerFwdBwd.statEmptyDiagnostics.status := 16#0000;
   instCmPusherRollerFwdBwd.statEmptyDiagnostics.subfunctionStatus := 16#0000;
   instCmPusherRollerFwdBwd.statEmptyDiagnostics.stateNumber := 0;
   instCmPusherRollerFwdBwd.instTimerReachPos.PT := T#0MS;
   instCmPusherRollerFwdBwd.instTimerReachPos.IN := FALSE;
   instCmPusherRollerFwdBwd.instTimerLeavePos.PT := T#0MS;
   instCmPusherRollerFwdBwd.instTimerLeavePos.IN := FALSE;
   instCmPusherRollerFwdBwd.instTimerDiscrepancyCheck.PT := T#0MS;
   instCmPusherRollerFwdBwd.instTimerDiscrepancyCheck.IN := FALSE;
   instCmPusherRollerFwdBwd.statDisableAlarms := FALSE;
   instCmPusherRollerFwdBwd.statDiagnostics.status := 16#7003;
   instCmPusherRollerFwdBwd.statDiagnostics.subfunctionStatus := 16#0000;
   instCmPusherRollerFwdBwd.statDiagnostics.stateNumber := 0;
   instCmPusherRollerFwdBwd.statEnablePrevious := TRUE;
   instCmPusherRollerFwdBwd.statFirstCall := FALSE;
   instCmPusherRollerFwdBwd.statResetPrevious := FALSE;
   instCmPusherRollerFwdBwd.statValid := TRUE;
   instCmPusherRollerFwdBwd.statBusy := TRUE;
   instCmPusherRollerFwdBwd.statError := FALSE;
   instCmPusherRollerFwdBwd.statInterlockWorkOff := FALSE;
   instCmPusherRollerFwdBwd.statInterlockHomeOff := FALSE;
   instCmPusherRollerFwdBwd.statFbState := 50;
   instCmPusherRollerFwdBwd.statFbStatePrevious := 50;
   instCmPusherRollerFwdBwd.statErrorUserCleared := FALSE;
   instCmPusherRollerFwdBwd.statErrorAutoCleared := FALSE;
   instCmPusherRollerFwdBwd.statErrorState := 16#0000;
   instCmPusherRollerFwdBwd.statDisablingCompleted := FALSE;
   instCmPusherRollerFwdBwd.statFeedbackHomePos := FALSE;
   instCmPusherRollerFwdBwd.statFeedbackWorkPos := FALSE;
   instManageAlarms.proDiagState.Total_Number := 487;
   instManageAlarms.proDiagState.All := TRUE;
   instManageAlarms.proDiagState.O := FALSE;
   instManageAlarms.proDiagState.I := FALSE;
   instManageAlarms.proDiagState.R := FALSE;
   instManageAlarms.proDiagState."A" := FALSE;
   instManageAlarms.proDiagState.P := FALSE;
   instManageAlarms.proDiagState.Merr := TRUE;
   instManageAlarms.proDiagState.Mtxt := FALSE;
   instManageAlarms.proDiagState.SV_Types := 16#20;
   instManageAlarms.proDiagState.C1 := TRUE;
   instManageAlarms.proDiagState.C2 := FALSE;
   instManageAlarms.proDiagState.C3 := FALSE;
   instManageAlarms.proDiagState.C4 := FALSE;
   instManageAlarms.proDiagState.C5 := FALSE;
   instManageAlarms.proDiagState.C6 := FALSE;
   instManageAlarms.proDiagState.C7 := FALSE;
   instManageAlarms.proDiagState.C8 := FALSE;
   instManageAlarms.proDiagState.Categories := 16#01;
   instManageAlarms.proDiagState.Sub_Cat_1 := 16#0000_0001;
   instManageAlarms.proDiagState.Sub_Cat_2 := 16#0000_0000;
   instManageAlarms.proDiagState.Reserved := 16#00;
   instManageAlarms.parentAlarmDB.error := TRUE;
   instManageAlarms.parentAlarmDB.warning := FALSE;
   instManageAlarms.parentAlarmDB.info := FALSE;
   instManageAlarms.alarmDB.error := TRUE;
   instManageAlarms.alarmDB.warning := FALSE;
   instManageAlarms.alarmDB.info := FALSE;
   instManageAlarms.hmiInterfaceDB.error := TRUE;
   instManageAlarms.hmiInterfaceDB.warning := FALSE;
   instManageAlarms.hmiInterfaceDB.info := FALSE;
   statUnitStatus.acknowledgeActive := FALSE;
   statUnitStatus.alarmsDisabled := FALSE;
   statUnitStatus.simulationActive := FALSE;
   statUnitStatus.safetyReleased := TRUE;
   statUnitStatus.state.current := 2;
   statUnitStatus.state.clearing := FALSE;
   statUnitStatus.state.stopped := TRUE;
   statUnitStatus.state.starting := FALSE;
   statUnitStatus.state.idle := FALSE;
   statUnitStatus.state.suspended := FALSE;
   statUnitStatus.state.execute := FALSE;
   statUnitStatus.state.stopping := FALSE;
   statUnitStatus.state.aborting := FALSE;
   statUnitStatus.state.aborted := FALSE;
   statUnitStatus.state.holding := FALSE;
   statUnitStatus.state.held := FALSE;
   statUnitStatus.state.unholding := FALSE;
   statUnitStatus.state.suspending := FALSE;
   statUnitStatus.state.unsuspending := FALSE;
   statUnitStatus.state.resetting := FALSE;
   statUnitStatus.state.completing := FALSE;
   statUnitStatus.state.complete := FALSE;
END_DATA_BLOCK
